FUNCTION_BLOCK FBUSER
VAR_INPUT
END_VAR
VAR_OUTPUT
END_VAR
VAR
END_VAR

END_FUNCTION_BLOCK

(* stored: Version 1.1.0.1, ProductVersion 3.1.4026.18
   POU FBUSER: Id {12916304-dbd3-450d-9ff6-e416bb8958dc}, SpecialFunc None *)
